FUNCTION Updete_Motor_Parameters_Reference
VAR_INPUT
	bUpdateValue : BOOL;
	fNewValue : REAL;
	stMotorParameters : REFERENCE TO ST_Motor;
END_VAR
VAR
END_VAR

IF bUpdateValue = 1 THEN
	stMotorParameters.fSpeedMax := fNewValue;
ELSE
	stMotorParameters.fSpeedMax := stMotorParameters.fSpeedMax;
END_IF

END_FUNCTION

(* stored: Version 1.1.0.1, ProductVersion 3.1.4024.12
   POU Updete_Motor_Parameters_Reference: Id {34ed5731-b12d-40f6-a8f6-9c9b7a879187}, SpecialFunc None *)
